{attribute addProperty BoxType "EP2316-0008-0016"}
{attribute addProperty Id "OutputAT %Q*ARRAY[0 ..7] OF BOOL6480"}
{attribute addProperty CRC "1062725746"}
{attribute addProperty SizeInBites "64"}
{attribute addProperty SizeInBytes "8"}
TYPE DO_Outputs_33B76376 :
STRUCT
	{attribute addProperty Name "Output"}
	Output AT %Q* : ARRAY[0 ..7] OF BOOL;
END_STRUCT
END_TYPE

(* stored: Version 1.2.0.0, ProductVersion 3.1.4024.9
   DUT DO_Outputs_33B76376: Id {ca6396db-038e-4f58-b65c-17ae4b3b6c00} *)
